FUNCTION FUN_AryBitCount_RD : UINT
VAR_IN_OUT
 IN : ARRAY[*] OF BOOL;
END_VAR
VAR  
  index : INT;
END_VAR

FUN_AryBitCount_RD:=0;
FOR index:=0 TO SIZEOF(IN)-1 DO
	IF IN[index] THEN
    FUN_AryBitCount_RD := FUN_AryBitCount_RD +1 ;
	END_IF;	
END_FOR;

END_FUNCTION

(* stored: Version 1.1.0.1, ProductVersion 3.1.4024.12
   POU FUN_AryBitCount_RD: Id {fd858496-4482-4ac4-aa76-d101a0e862b0}, SpecialFunc None *)
